// TwinCAT 3 PLC project PLC
// ProgramVersion: 3.1.4024.0
// libraries:
//   Tc2_Standard, * (Beckhoff Automation GmbH)
//   Tc2_System, * (Beckhoff Automation GmbH)
//   Tc3_Module, * (Beckhoff Automation GmbH)
// project tree:
//   / GlobalTextList.TcGTLO, PlcTask.TcTTO, Visualization Manager.TcVMO (not stored)
//   POUs/ MAIN.TcPOU, Q10.TcPOU, Q1.TcPOU, Q2.TcPOU, Q3.TcPOU, Q4.TcPOU, Q5.TcPOU, Q6.TcPOU, Q7.TcPOU, Q8.TcPOU, Q9.TcPOU
//   VISUs/ Visualization.TcVIS
// real-time tasks:
//   TASK PlcTask: cycle T#10ms, priority 20, ADS port 350

CONFIGURATION PLC
    RESOURCE PLC ON TwinCAT3
        TASK PlcTask(INTERVAL := T#10ms, PRIORITY := 20);
        PROGRAM MAIN WITH PlcTask : MAIN;
    END_RESOURCE
END_CONFIGURATION

// ---- POUs/MAIN.TcPOU
PROGRAM MAIN
VAR
END_VAR

Q10();

END_PROGRAM

// ---- POUs/Q10.TcPOU
PROGRAM Q10
VAR
	extrude		: BOOL	:= FALSE;
	extruding 	: BOOL 	:= FALSE;
	extruded	: BOOL	:= FALSE;
	warning		: BOOL	:= FALSE;
	TON_0: TON;
	
	count_i		: UINT	:=0;
	count_t		: TIME	:= T#0S;
END_VAR

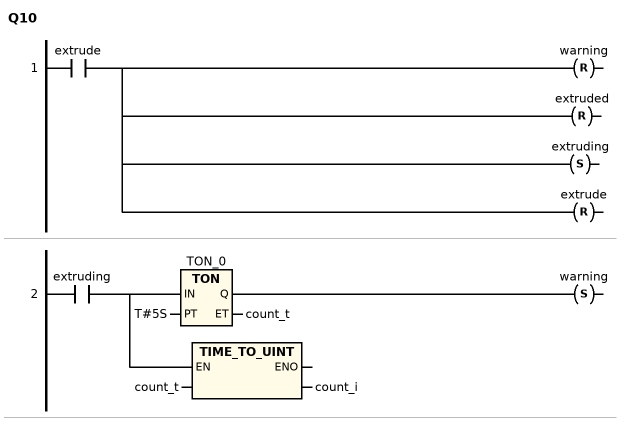
// NETWORK 1
warning R= extrude;
extruded R= extrude;
extruding S= extrude;
extrude R= extrude;

// NETWORK 2
TON_0(IN := extruding, PT := T#5S, ET => count_t); // TON
warning S= TON_0.Q;
IF extruding THEN count_i := TIME_TO_UINT(count_t); END_IF

END_PROGRAM

// ---- POUs/Q1.TcPOU
PROGRAM Q1
VAR
	loop : INT := 1;
END_VAR

END_PROGRAM

// ---- POUs/Q2.TcPOU
PROGRAM Q2
VAR
	tempurature : REAL := 26.5;
END_VAR

END_PROGRAM

// ---- POUs/Q3.TcPOU
PROGRAM Q3
VAR
	// INT : num1 := 1;
	// DataType and VarName are wrong way round
	num1 : INT := 1;
END_VAR

END_PROGRAM

// ---- POUs/Q4.TcPOU
PROGRAM Q4
VAR
	// num1 := 1;
	// Missing DataType
	num1 : INT := 1;
END_VAR

END_PROGRAM

// ---- POUs/Q5.TcPOU
PROGRAM Q5
VAR
	num1 : INT := 1;
 	num2 : INT := 2;
 	res : INT := 0;
	op1: INT;
	op2: INT;
END_VAR

op1 := num1;
op2 := num2;
res := op1 / op2 - 5;

// To run, paste "Q5();" into the MAIN proram
// Result: res == -5
// 1 / 2 = 0.5 -> 0
// 0 - 5 = -5

END_PROGRAM

// ---- POUs/Q6.TcPOU
PROGRAM Q6
VAR
	A : BOOL := TRUE;
	B : BOOL := FALSE;
	C : BOOL := FALSE;
END_VAR

// Result: C == TRUE

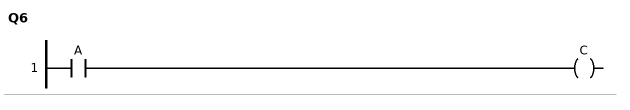
// NETWORK 1
C := A;

END_PROGRAM

// ---- POUs/Q7.TcPOU
PROGRAM Q7
VAR
	 A : BOOL := TRUE;
 B : BOOL := FALSE;
 C : BOOL := FALSE;
END_VAR

// Result: C == TRUE;

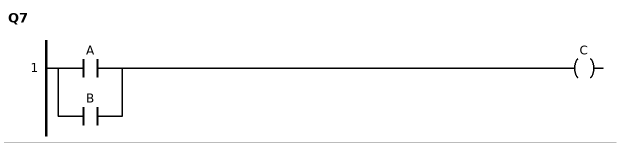
// NETWORK 1
C := A OR B;

END_PROGRAM

// ---- POUs/Q8.TcPOU
PROGRAM Q8
VAR
	input : BOOL;
	output: BOOL;
END_VAR

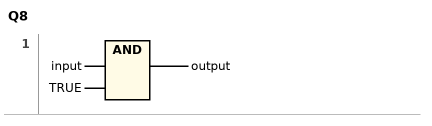
// NETWORK 1
output := input AND TRUE;

END_PROGRAM

// ---- POUs/Q9.TcPOU
PROGRAM Q9
VAR
	inputButton : BOOL := FALSE;
	inputReset	: BOOL := FALSE;
		
	timerStart	: BOOL := FALSE;
	timerRunning: BOOL := FALSE;
	Timer_On: TON;	
	timerCount	: TIME := T#0S;
	
	warning		: BOOL := FALSE;
	count_warn	: TIME := T#10S;
	output		: BOOL := FALSE;
	count_out	: TIME := T#15S;

END_VAR
VAR // added by the converter: edge detectors and wires of the graphical bodies
    _w1, _w2, _w3, _w4 : BOOL;
END_VAR

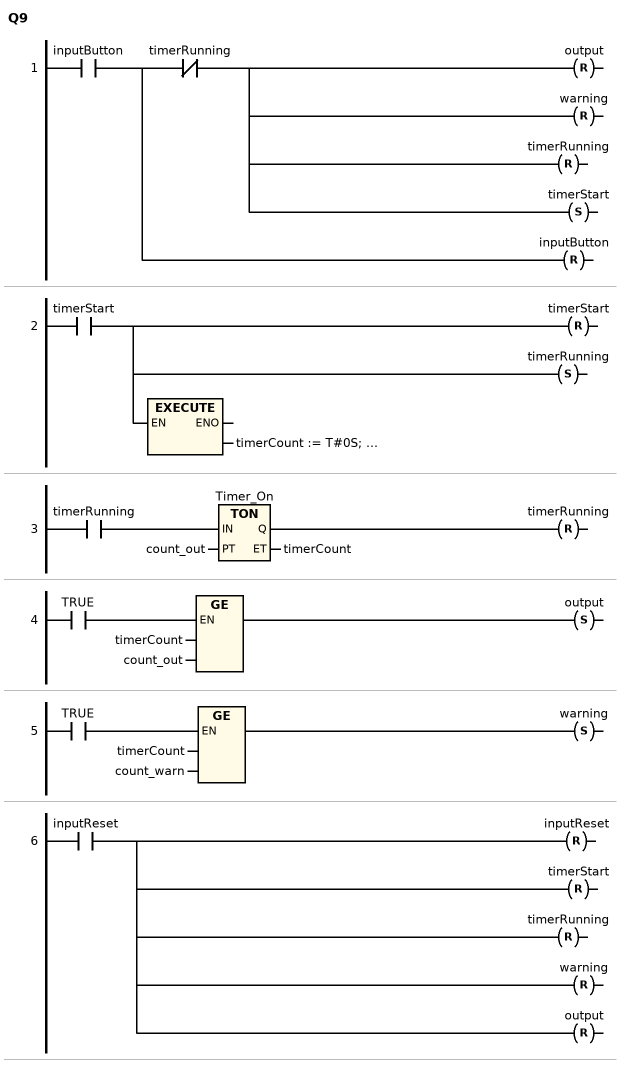
// NETWORK 1
_w1 := inputButton;
_w2 := _w1 AND NOT timerRunning;
output R= _w2;
warning R= _w2;
timerRunning R= _w2;
timerStart S= _w2;
inputButton R= _w1;

// NETWORK 2
_w3 := timerStart;
timerStart R= _w3;
timerRunning S= _w3;
IF _w3 THEN timerCount := T#0S; END_IF

// NETWORK 3
Timer_On(IN := timerRunning, PT := count_out, ET => timerCount); // TON
timerRunning R= Timer_On.Q;

// NETWORK 4
output S= timerCount >= count_out;

// NETWORK 5
warning S= timerCount >= count_warn;

// NETWORK 6
_w4 := inputReset;
inputReset R= _w4;
timerStart R= _w4;
timerRunning R= _w4;
warning R= _w4;
output R= _w4;

END_PROGRAM

// ---- GlobalTextList.TcGTLO
TEXTLIST GlobalTextList
  772 = 'Extrude'
  715 = 'Extruded'
  354 = 'Extruding'
  72 = 'Inpaut'
  571 = 'Input'
  117 = 'Output'
  153 = 'Status'
  411 = 'Warning'
END_TEXTLIST

// ---- VISUs/Visualization.TcVIS
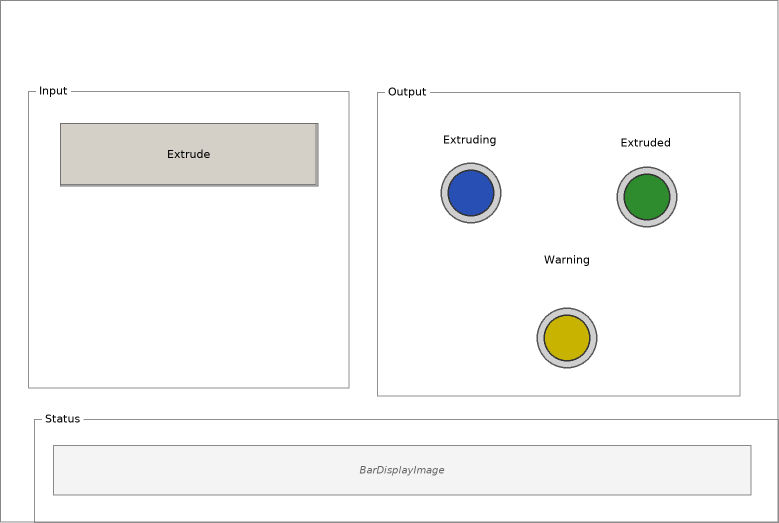
VISUALIZATION Visualization  // 779x523
    GroupBox (28,83 321x305), "Input"
        Button (32,40 258x63), "Extrude"
            OnMouseClick: execute { Q10.extrude := TRUE; }
    GroupBox (377,84 363x312), "Output"
        Lamp1 (59,74 70x70), variable: Q10.extruding, style: Lamp-Lamp1-Blue
        Lamp1 (155,219 70x70), variable: Q10.warning, style: Lamp-Lamp1-Yellow
        Label (18,41 150x30), "Extruding"
        Label (194,44 150x30), "Extruded"
        Label (115,161 150x30), "Warning"
        Lamp1 (235,78 70x70), variable: Q10.extruded, style: Lamp-Lamp1-Green
    GroupBox (34,411 745x112), "Status"
        BarDisplayImage (19,34 698x50), value: Q10.count_i, style: BarDisplayImage-Gray, scale format: %.1f, scale 0..20000
END_VISUALIZATION
